// TIA Portal V20 export
DATA_BLOCK "LBP_TMSpindle"   // DB72
TITLE = Tool management / Gestion des outils
{ S7_Optimized_Access := 'FALSE' }
AUTHOR : SINUMERIK
FAMILY : SINUMERIK_ONE
VERSION : 6.24
// Interface between user program and tool management, contains signals for spindle as change position. / Interface entre programme utilisateur et gestion d'outil, contient des signaux pour broche en tant que position de changement.
// stored: AutoNumber false, InstanceOfName LBP_typeTMSpindle, InstanceOfType UDT
"LBP_typeTMSpindle"
   // VAR RETAIN
   //    IFNo : Array[1..16] of Bool;
   //    Quit : Array[1..16] of Bool;
   //    TIF : Array[1..16] of Struct
   //       Comp : Bool;
   //       Perform : Bool;
   //       Prepare : Bool;
   //       T0 : Bool;
   //       OldTinDBW42 : Bool;
   //       ManTIn : Bool;
   //       ManTOut : Bool;
   //       SpiTRSpi : Bool;
   //       PerfStatusError : Bool;
   //       n1_1 : Bool;
   //       n1_2 : Bool;
   //       n1_3 : Bool;
   //       n1_4 : Bool;
   //       n1_5 : Bool;
   //       n1_6 : Bool;
   //       DataInDB1072 : Bool;
   //       Channel : Byte;
   //       TMNo : Byte;
   //       VdiTcp0 : DInt;
   //       VdiTcp1 : DInt;
   //       VdiTcp2 : DInt;
   //       BufferIdent : Int;
   //       BufferNo : Int;
   //       SMag : Int;
   //       SLoc : Int;
   //       TMag : Int;
   //       TLoc : Int;
   //       LocType : Int;
   //       SLeft : Int;
   //       SRight : Int;
   //       STop : Int;
   //       SBottom : Int;
   //       TInBuffer : Bool;
   //       IgnoreDisabled : Bool;
   //       Unload : Bool;
   //       Load : Bool;
   //       MasterTool : Bool;
   //       n38_5 : Bool;
   //       Exchange_1to1 : Bool;
   //       HandTool : Bool;
   //       Active : Bool;
   //       Enabled : Bool;
   //       Disabled : Bool;
   //       Measured : Bool;
   //       Prewarn : Bool;
   //       Change : Bool;
   //       FixedLoc : Bool;
   //       Used : Bool;
   //       TNo : Int;
   //       OldTBufferNo : Int;
   //       MyMag : Int;
   //       MyPlace : Int;
   //    END_STRUCT;
   // END_VAR
BEGIN
END_DATA_BLOCK
